// TIA Portal V20 export
DATA_BLOCK "InstGetAxisStatus"   // DB198
AUTHOR : Siemens Digital Industries
FAMILY : LAF
NAME : LAF_GetAxisStatus
VERSION : 1.1
// stored: InstanceOfName LAF_GetAxisStatus, InstanceOfType FB
"LAF_GetAxisStatus"
   // VAR_INPUT
   //    enable : Bool;
   // END_VAR
   // VAR_OUTPUT
   //    valid { ExternalWritable := 'False'} : Bool;
   //    busy { ExternalWritable := 'False'} : Bool;
   //    error { ExternalWritable := 'False'} : Bool;
   //    status { ExternalWritable := 'False'} : Word;
   //    diagnostics { ExternalWritable := 'False'} : "LAF_typeDiagnostics";
   // END_VAR
   // VAR_IN_OUT
   //    configuration : Array[*] of "LAF_typeDriveDiagConfig";
   //    moduleInterface : "LAF_typeDriveDiagInterfaceHmi";
   // END_VAR
   // VAR
   //    statInternal { ExternalAccessible := 'False'; ExternalVisible := 'False'; ExternalWritable := 'False'} : Struct
   //       enablePrevious : Bool;
   //       valid : Bool;
   //       busy : Bool;
   //       error : Bool;
   //       errorUserCleared : Bool;
   //       errorAutoCleared : Bool;
   //       disablingCompleted : Bool;
   //       diagnostics : "LAF_typeDiagnostics";
   //       emptyDiagnostics : "LAF_typeDiagnostics";
   //    END_STRUCT;
   //    statMainState { ExternalAccessible := 'False'; ExternalVisible := 'False'; ExternalWritable := 'False'} : DInt;
   //    statArrayMin { ExternalAccessible := 'False'; ExternalVisible := 'False'; ExternalWritable := 'False'} : DInt;
   //    statArrayMax { ExternalAccessible := 'False'; ExternalVisible := 'False'; ExternalWritable := 'False'} : DInt;
   // END_VAR
BEGIN
END_DATA_BLOCK
